// TIA Portal V19 export
DATA_BLOCK "PPrgArchive14"   // DB513
// stored: IsOnlyStoredInLoadMemory true, MemoryReserve 0, Namespace G
   VAR RETAIN
      PRG : Array[1301..1400] of "PPrg_Data";
   END_VAR
BEGIN
END_DATA_BLOCK
